TYPE ST_DoDi :
STRUCT	
	input	: ST_DoDi_in;	
	
	output	: ST_DoDi_out;	
END_STRUCT
END_TYPE

(* stored: Version 1.1.0.1, ProductVersion 3.1.4024.9
   DUT ST_DoDi: Id {eea794f4-b79c-40c6-8283-a801508611e1} *)
